FUNCTION_BLOCK ABSTRACT PAC_MoveWorkpiece_Base EXTENDS ControlPrimitiveBase
VAR_INPUT
END_VAR
VAR_OUTPUT
END_VAR
VAR
	m_ptrPAC: POINTER TO PicAlphaConveyor;
	
	m_step: INT := 0;
END_VAR

SUPER^();

METHOD  Abort : BOOL
VAR_INPUT
END_VAR
m_ptrPAC^.METH_ConveyorStop();
m_ptrPAC^.METH_Switch_Retract();
Abort := TRUE;
END_METHOD

METHOD PROTECTED ABSTRACT AtTarget : BOOL
VAR_INPUT
END_VAR
END_METHOD

METHOD PROTECTED ABSTRACT EjectOperation : BOOL
VAR_INPUT
END_VAR
END_METHOD

(* Execution logic of this Control Primitive. *)
METHOD PROTECTED ExecuteInternal : BOOL
VAR_INPUT
	i_params: ParameterSet;
END_VAR
CASE m_step OF
	0: // to target	
	IF NOT AtTarget() THEN
		m_ptrPAC^.METH_ConveyorForward();
		m_step := 1;
	END_IF
		
	1:
	IF AtTarget() THEN
		m_ptrPAC^.METH_ConveyorStop();
		//m_ptrPAC^.METH_Switch_Extend();
		m_step := 2;
	END_IF
	
	2:
	IF EjectOperation() THEN
		m_step := 0;
		ExecuteInternal := TRUE;
	END_IF
		
END_CASE
END_METHOD

END_FUNCTION_BLOCK

(* stored: Version 1.1.0.1, ProductVersion 3.1.4024.12
   POU PAC_MoveWorkpiece_Base: Id {a028fe99-a406-423b-81fa-142d041a937b}, SpecialFunc None
   Method Abort: Id {835a33f6-5d18-4808-9533-0a62672b4ac0}
   Method AtTarget: Id {ad66d4b4-0b80-48ef-8921-dba0e78cb219}
   Method EjectOperation: Id {fe1251da-1d05-406f-b4db-65d2fd4adbd0}
   Method ExecuteInternal: Id {08fcb40a-0998-4cda-bce6-29c79df8925d} *)
